/// GearIn parameter strucure
TYPE ST_AxisGearInParameter :
STRUCT
	eMasterId: E_Axis;
	fbMaster: REFERENCE TO AXIS_REF;
	fGearRatio: LREAL;
	fAcceleration: LREAL;
	fDeceleration: LREAL;
	fJerk: LREAL;
	eBufferMode: MC_BufferMode;
	stOptions: ST_GearInDynOptions;
END_STRUCT
END_TYPE

(* stored: Version 1.1.0.1, ProductVersion 3.1.4020.12
   DUT ST_AxisGearInParameter: Id {0afffcf3-dccc-4b56-b924-948f7c2ed290} *)
